// TIA Portal V19 export
DATA_BLOCK "AlarmBitScada"   // DB25
{ S7_Optimized_Access := 'TRUE' }
AUTHOR : FLA
FAMILY : UHT
VERSION : 1.0
// stored: AutoNumber false, MemoryReserve 0
   VAR RETAIN
      A01_TankInProcess : Bool;   // PushButtonAlarm
      A02_TankNotClean : Bool;   // PushButtonAlarm
      A03_NoInstrumentAir : Bool;   // PushButtonAlarm
      A04_NoSteam : Bool;   // PushButtonAlarm
      A05_DrainIsActive : Bool;   // PushButtonAlarm
      A06_CipFillerStarted : Bool;   // PushButtonAlarm
      A07_CipUnitOccupied : Bool;   // PushButtonAlarm
      A08_NotReadyForCip : Bool;   // PushButtonAlarm
      A09_NoProcessActive : Bool;   // PushButtonAlarm
      A10_AllreadyInStopPhase : Bool;   // PushButtonAlarm
      A11_TankIsBeingFilled : Bool;   // PushButtonAlarm
      A12_NotReadyForTotalStop : Bool;   // PushButtonAlarm
      A13_DrainTankNotAllowed : Bool;   // PushButtonAlarm
      A14_CipOnTankStared : Bool;   // PushButtonAlarm
      A15_ChainWashSelected : Bool;   // PushButtonAlarm
      A16_NoCipProgramSelected : Bool;   // PushButtonAlarm
      A17_ContinueDosingSelect : Bool;   // PushButtonAlarm
      A18 : Bool;   // PushButtonAlarm
      A19 : Bool;   // PushButtonAlarm
      A20 : Bool;   // PushButtonAlarm
      A21 : Bool;   // PushButtonAlarm
      A22 : Bool;   // PushButtonAlarm
      A23 : Bool;   // PushButtonAlarm
      A24 : Bool;   // PushButtonAlarm
      A25 : Bool;   // PushButtonAlarm
      A26 : Bool;   // PushButtonAlarm
      A27 : Bool;   // PushButtonAlarm
      A28 : Bool;   // PushButtonAlarm
      A29 : Bool;   // PushButtonAlarm
      A30 : Bool;   // PushButtonAlarm
      A31 : Bool;   // PushButtonAlarm
      A32 : Bool;   // PushButtonAlarm
      A33_TT0176TooLow : Bool;   // ProcessAlarm
      A34_TT0160TooLow : Bool;   // ProcessAlarm
      A35_TT0163TooLow : Bool;   // ProcessAlarm
      A36_TT0178TooLow : Bool;   // ProcessAlarm
      A37_TT0176Low : Bool;   // ProcessAlarm
      A38_TT0178Low : Bool;   // ProcessAlarm
      A39_TankReadyforProd : Bool;   // ProcessAlarm
      A40_LyedosingTooLong : Bool;   // ProcessAlarm
      A41_AcidDosingTooLong : Bool;   // ProcessAlarm
      A42_DrainTheTank : Bool;   // ProcessAlarm
      A43_WaitingForCipUnit : Bool;   // ProcessAlarm
      A44_FillPressureTooLow : Bool;   // ProcessAlarm
      A45_FillingPressureLow : Bool;   // ProcessAlarm
      A46_LyeContainerEmpty : Bool;   // ProcessAlarm
      A47_AcidContainerEmpty : Bool;   // ProcessAlarm
      A48_TankEmpty : Bool;   // ProcessAlarm
      A49_TankFull : Bool;   // ProcessAlarm
      A50_SiemensBatteryLow : Bool;   // ProcessAlarm
      A51_NoWater : Bool;   // ProcessAlarm
      A52_ProdAtFillingMash : Bool;   // ProcessAlarm
      A53_FillerNotReadyForCip : Bool;   // ProcessAlarm
      A54_NoInstrumentAir : Bool;   // ProcessAlarm
      A55_NoSteam : Bool;   // ProcessAlarm
      A56 : Bool;   // ProcessAlarm
      A57_TT0951TooLow : Bool;   // ProcessAlarm
      A58_TT0951Low : Bool;   // ProcessAlarm
      A59_TT0950TooLow : Bool;   // ProcessAlarm
      A60_TT0950Low : Bool;   // ProcessAlarm
      A61_Hamba_Valve_Fault : Bool;   // ProcessAlarm
      A62_Hamba_Barrier_low : Bool;   // ProcessAlarm
      A63_Stop_CIP_PB_Operated : Bool;   // ProcessAlarm
      A64_TT0178_High : Bool;   // Condensate temperature High
      A65_TT0930_Low : Bool;   // TT0930 Low Production
      A66_TT0930_Low_SIP : Bool;   // TT0930 Low SIP
      A67_TT0931_Low : Bool;   // TT0931 Low Production
      A68_CT0930_High : Bool;   // CT0930 High Conductivity - suspect V01.01 Seals
      dx8_4_Spare : Bool;   // ProcessAlarm
      dx8_5_Spare : Bool;   // ProcessAlarm
      dx8_6_Spare : Bool;   // ProcessAlarm
      dx8_7_Spare : Bool;   // ProcessAlarm
      dx9_0_Spare : Bool;   // ProcessAlarm
      dx9_1_Spare : Bool;   // ProcessAlarm
      dx9_2_Spare : Bool;   // ProcessAlarm
      dx9_3_Spare : Bool;   // ProcessAlarm
      dx9_4_Spare : Bool;   // ProcessAlarm
      dx9_5_Spare : Bool;   // ProcessAlarm
      dx9_6_Spare : Bool;   // ProcessAlarm
      dx9_7_Spare : Bool;   // ProcessAlarm
      dx10_0_Spare : Bool;   // ProcessAlarm
      dx10_1_Spare : Bool;   // ProcessAlarm
      dx10_2_Spare : Bool;   // ProcessAlarm
      dx10_3_Spare : Bool;   // ProcessAlarm
      dx10_4_Spare : Bool;   // ProcessAlarm
      dx10_5_Spare : Bool;   // ProcessAlarm
      dx10_6_Spare : Bool;   // ProcessAlarm
      dx10_7_Spare : Bool;   // ProcessAlarm
      dx11_0_Spare : Bool;   // ProcessAlarm
      dx11_1_Spare : Bool;   // ProcessAlarm
      dx11_2_Spare : Bool;   // ProcessAlarm
      dx11_3_Spare : Bool;   // ProcessAlarm
      dx11_4_Spare : Bool;   // ProcessAlarm
      dx11_5_Spare : Bool;   // ProcessAlarm
      dx11_6_Spare : Bool;   // ProcessAlarm
      dx11_7_Spare : Bool;   // ProcessAlarm
   END_VAR
BEGIN
END_DATA_BLOCK
